(* Logix 5000 project; controller DC01 vendor 1 type 14 code 165 rev 32.12; software revision 32.04; part 9 of 13 *)
(* tags used below, declared in another part *)
   Always_Off : BOOL;
   Break_1stStation : BOOL;
   Break_LineWide : BOOL;
   Break_WorkCenter : BOOL;
   Break_Workstation : BOOL;
   FaultExists : CONTROL;
   LN03_MainLine_MSG : MESSAGE;   // Data Messages From Assembly Line 3 To Data Concentrator 1
   Local_Timer : TIMER[30];
   ONS_0 : DINT;
   Scheduled_Units_Buffer : DINT;
   Shift_Reset : BOOL;
   Shift_Reset_ONS : BOOL;
   LN02_Schedule : UDT_Current_Status;
   LN03_1st_Station_Break_Code : DINT;
   LN03_Additional_Break_Limit_Mins : DINT;
   LN03_Boxing_MNT : DINT;
   LN03_Console_MNT : DINT;
   LN03_Cooktop_MNT : DINT;
   LN03_Current_Shift_Duration_Mins : DINT;   // CURRENT SHIFT TOTAL MINUTES SCHEDULED
   LN03_Current_Shift_Duration_wBreaks_Mins : DINT;
   LN03_DC_Controlled_Theoretical_Units : BOOL;
   LN03_Door_MNT : DINT;
   LN03_FPY : REAL;
   LN03_FrontFrame_MNT : DINT;
   LN03_Ignition_NewSNModel : BOOL[32];
   LN03_Ignition_SNModelMSG : STRING[5];
   LN03_LeakTest_MNT : DINT;
   LN03_MachineOverAll_MNT : DINT;
   LN03_Main_Messages : DINT[250];
   LN03_MainBack_MNT : DINT;
   LN03_Messages_Barcode_SNModel : Barcode_SNModel;
   LN03_OT_Shift_Break_In_Minutes : DINT;
   LN03_OvenCavity_MNT : DINT;
   LN03_Schedule : UDT_Current_Status;
   LN03_Schedule_Cycle_Timer : TIMER;   // UNIT CYCLE ( TAKT TIME ) TIMER
   LN03_Schedule_Max_Break_Duration : DINT;
   LN03_Schedule_Max_Break_Timer : TIMER;
   LN03_Schedule_TAKT : REAL;
   LN03_SidePanels_MNT : DINT;
   LN03_Standard_Shift_Break_In_Minutes : DINT;
   LN03_StorageDrawer_MNT : DINT;
   LN03_Test_MNT : DINT;
   LN03_Theoretical_Units_Counter : COUNTER;   // CURRENT NUMBER OF UNITS THAT SHOULD BE BUILT
   LN03_Theoretical_Units_Counter_ONS : BOOL;
   LN03_Units_for_repair : DINT;
   LN03_Wiring_MNT : DINT;
   LN03ECM01 : DINT;
   LN03ECM02 : DINT;
   LN03ECM03 : DINT;
   LN03ECM04 : DINT;
   LN03ECM06 : DINT;
   LN03EDM04 : DINT;
   LN03EEM01 : DINT;
   LN03EES02 : DINT;
   LN03EES03 : DINT;
   LN03EES04 : DINT;
   LN03EGM01 : DINT;
   LN03EGM02 : DINT;
   LN03EHM01 : DINT;
   LN03NAS01 : DINT;
   LN03NAS02 : DINT;
   LN03NAS03 : DINT;
   LN03NAS04 : DINT;
   LN03NBS03 : DINT;
   LN03NCS01 : DINT;
   LN03NCS02 : DINT;
   LN03NCS03 : DINT;
   LN03NCS04 : DINT;
   LN03NCS05 : DINT;
   LN03NFS01 : DINT;
   LN03NFS03 : DINT;
   LN03SBS01 : DINT;
   LN03SBS02 : DINT;
   LN03SBS03 : DINT;
   LN03SCS03 : DINT;
   LN03SES01 : DINT;
   LN03SFS01 : DINT;
   LN03SFS02 : DINT;
   LN03SFS03 : DINT;
   LN03SFS04 : DINT;
   LN03WAM01 : DINT;
   LN03WBM01 : DINT;
   LN03WBM02 : DINT;
   LN03WCM02 : DINT;
   LN03WCM03 : DINT;
   LN03WCM04 : DINT;
   LN03WCM05 : DINT;
   LN03WDM01 : DINT;
   LN03WDM02 : DINT;
   LN03WDM03 : DINT;
   LN03WDM04 : DINT;
   LN03WDM05 : DINT;
   LN03WEM01 : DINT;
   LN03WEM02 : DINT;
   LN03WFM01 : DINT;
   LN03WFM02 : DINT;
   LN03WFM03 : DINT;
   LN03WFM04 : DINT;
   LN03WFM05 : DINT;
   LN03WFM06 : DINT;
   LN03WGM01 : DINT;
(* LN03, continued *)

ROUTINE R02_CurrentShift_Calcs   (* ladder *)
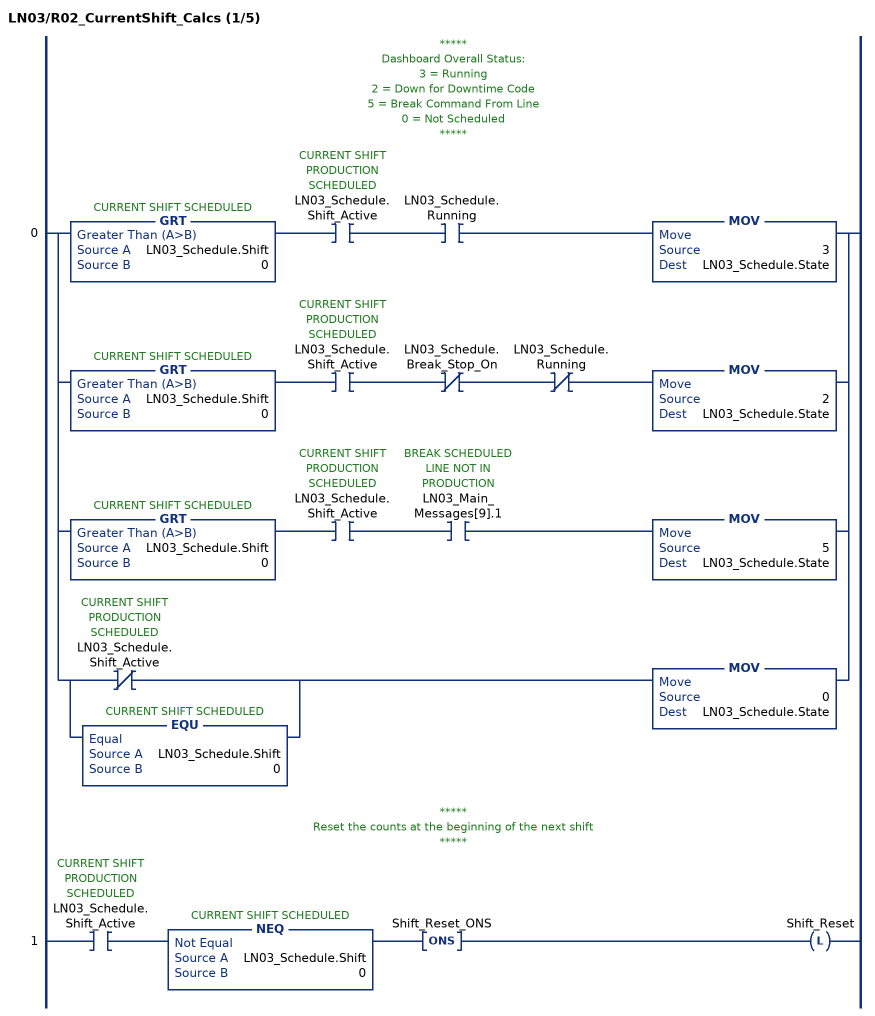
   // *****
   // Dashboard Overall Status:
   // 3 = Running
   // 2 = Down for Downtime Code
   // 5 = Break Command From Line
   // 0 = Not Scheduled
   // *****
   0: [GRT(LN03_Schedule.Shift,0) XIC(LN03_Schedule.Shift_Active) XIC(LN03_Schedule.Running) MOV(3,LN03_Schedule.State) ,GRT(LN03_Schedule.Shift,0) XIC(LN03_Schedule.Shift_Active) XIO(LN03_Schedule.Break_Stop_On) XIO(LN03_Schedule.Running) MOV(2,LN03_Schedule.State) ,GRT(LN03_Schedule.Shift,0) XIC(LN03_Schedule.Shift_Active) XIC(LN03_Main_Messages[9].1) MOV(5,LN03_Schedule.State) ,[XIO(LN03_Schedule.Shift_Active) ,EQU(LN03_Schedule.Shift,0) ] MOV(0,LN03_Schedule.State) ];
   // *****
   // Reset the counts at the beginning of the next shift
   // *****
   1: XIC(LN03_Schedule.Shift_Active)NEQ(LN03_Schedule.Shift,0)ONS(Shift_Reset_ONS)OTL(Shift_Reset);
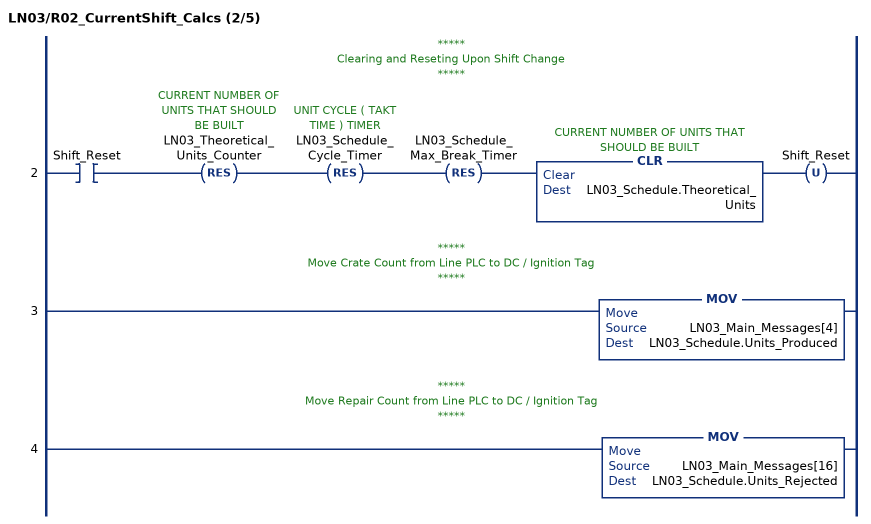
   // *****
   // Clearing and Reseting Upon Shift Change
   // *****
   2: XIC(Shift_Reset)RES(LN03_Theoretical_Units_Counter)RES(LN03_Schedule_Cycle_Timer)RES(LN03_Schedule_Max_Break_Timer)CLR(LN03_Schedule.Theoretical_Units)OTU(Shift_Reset);
   // *****
   // Move Crate Count from Line PLC to DC / Ignition Tag
   // *****
   3: MOV(LN03_Main_Messages[4],LN03_Schedule.Units_Produced);
   // *****
   // Move Repair Count from Line PLC to DC / Ignition Tag
   // *****
   4: MOV(LN03_Main_Messages[16],LN03_Schedule.Units_Rejected);
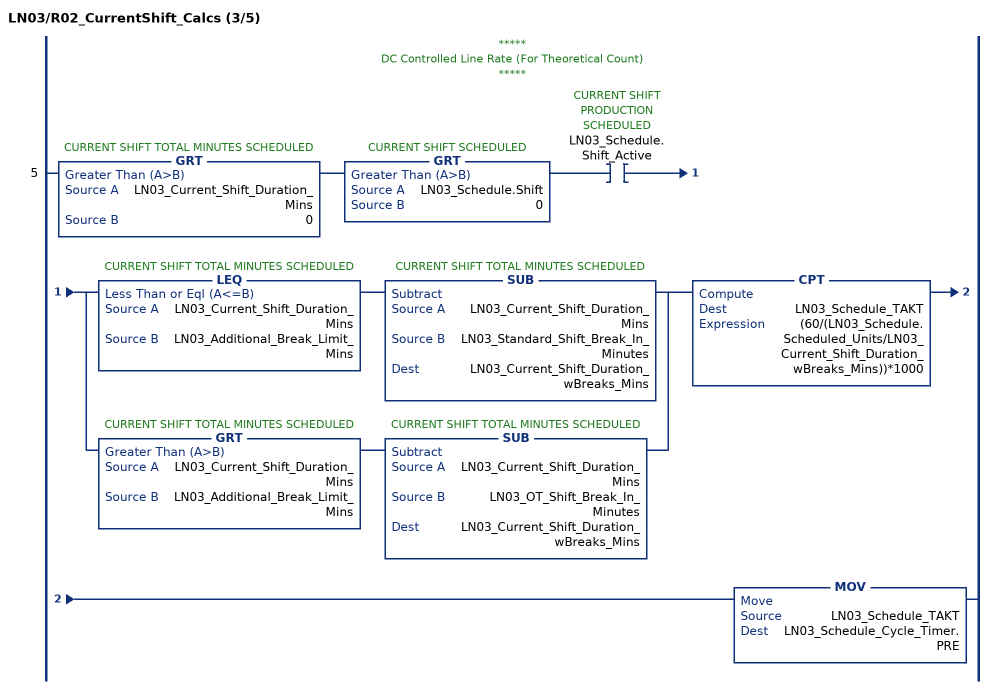
   // *****
   // DC Controlled Line Rate (For Theoretical Count)
   // *****
   5: GRT(LN03_Current_Shift_Duration_Mins,0)GRT(LN03_Schedule.Shift,0)XIC(LN03_Schedule.Shift_Active)[LEQ(LN03_Current_Shift_Duration_Mins,LN03_Additional_Break_Limit_Mins) SUB(LN03_Current_Shift_Duration_Mins,LN03_Standard_Shift_Break_In_Minutes,LN03_Current_Shift_Duration_wBreaks_Mins) ,GRT(LN03_Current_Shift_Duration_Mins,LN03_Additional_Break_Limit_Mins) SUB(LN03_Current_Shift_Duration_Mins,LN03_OT_Shift_Break_In_Minutes,LN03_Current_Shift_Duration_wBreaks_Mins) ]CPT(LN03_Schedule_TAKT,(60/(LN03_Schedule.Scheduled_Units/LN03_Current_Shift_Duration_wBreaks_Mins))*1000)MOV(LN03_Schedule_TAKT,LN03_Schedule_Cycle_Timer.PRE);
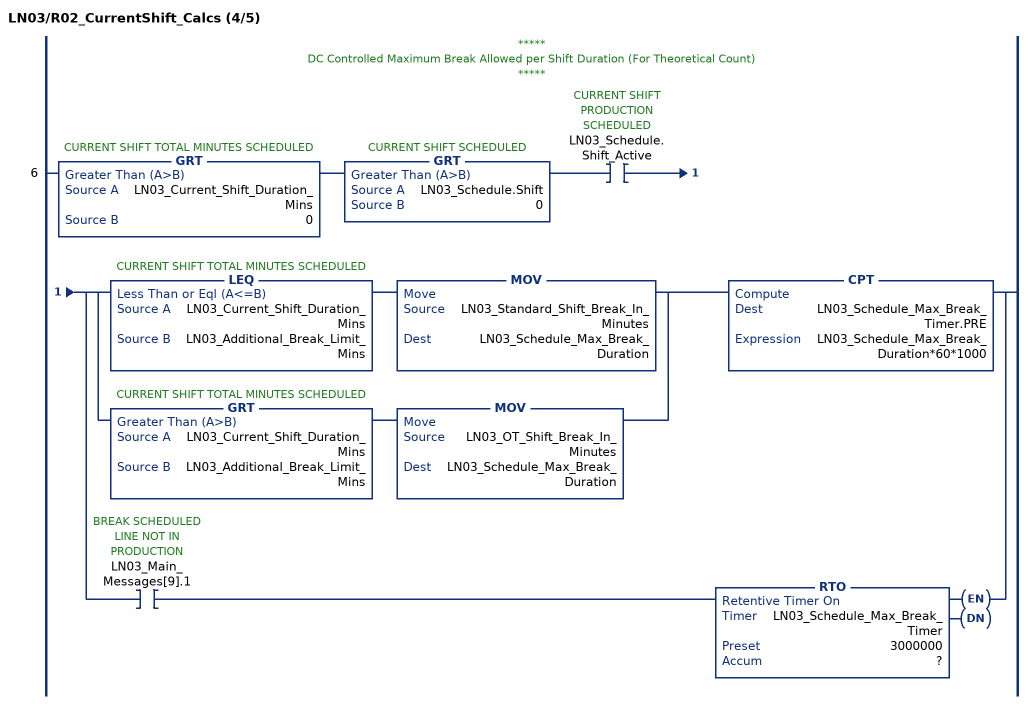
   // *****
   // DC Controlled Maximum Break Allowed per Shift Duration (For Theoretical Count)
   // *****
   6: GRT(LN03_Current_Shift_Duration_Mins,0)GRT(LN03_Schedule.Shift,0)XIC(LN03_Schedule.Shift_Active)[[LEQ(LN03_Current_Shift_Duration_Mins,LN03_Additional_Break_Limit_Mins) MOV(LN03_Standard_Shift_Break_In_Minutes,LN03_Schedule_Max_Break_Duration) ,GRT(LN03_Current_Shift_Duration_Mins,LN03_Additional_Break_Limit_Mins) MOV(LN03_OT_Shift_Break_In_Minutes,LN03_Schedule_Max_Break_Duration) ] CPT(LN03_Schedule_Max_Break_Timer.PRE,LN03_Schedule_Max_Break_Duration*60*1000) ,XIC(LN03_Main_Messages[9].1) RTO(LN03_Schedule_Max_Break_Timer,?,?) ];
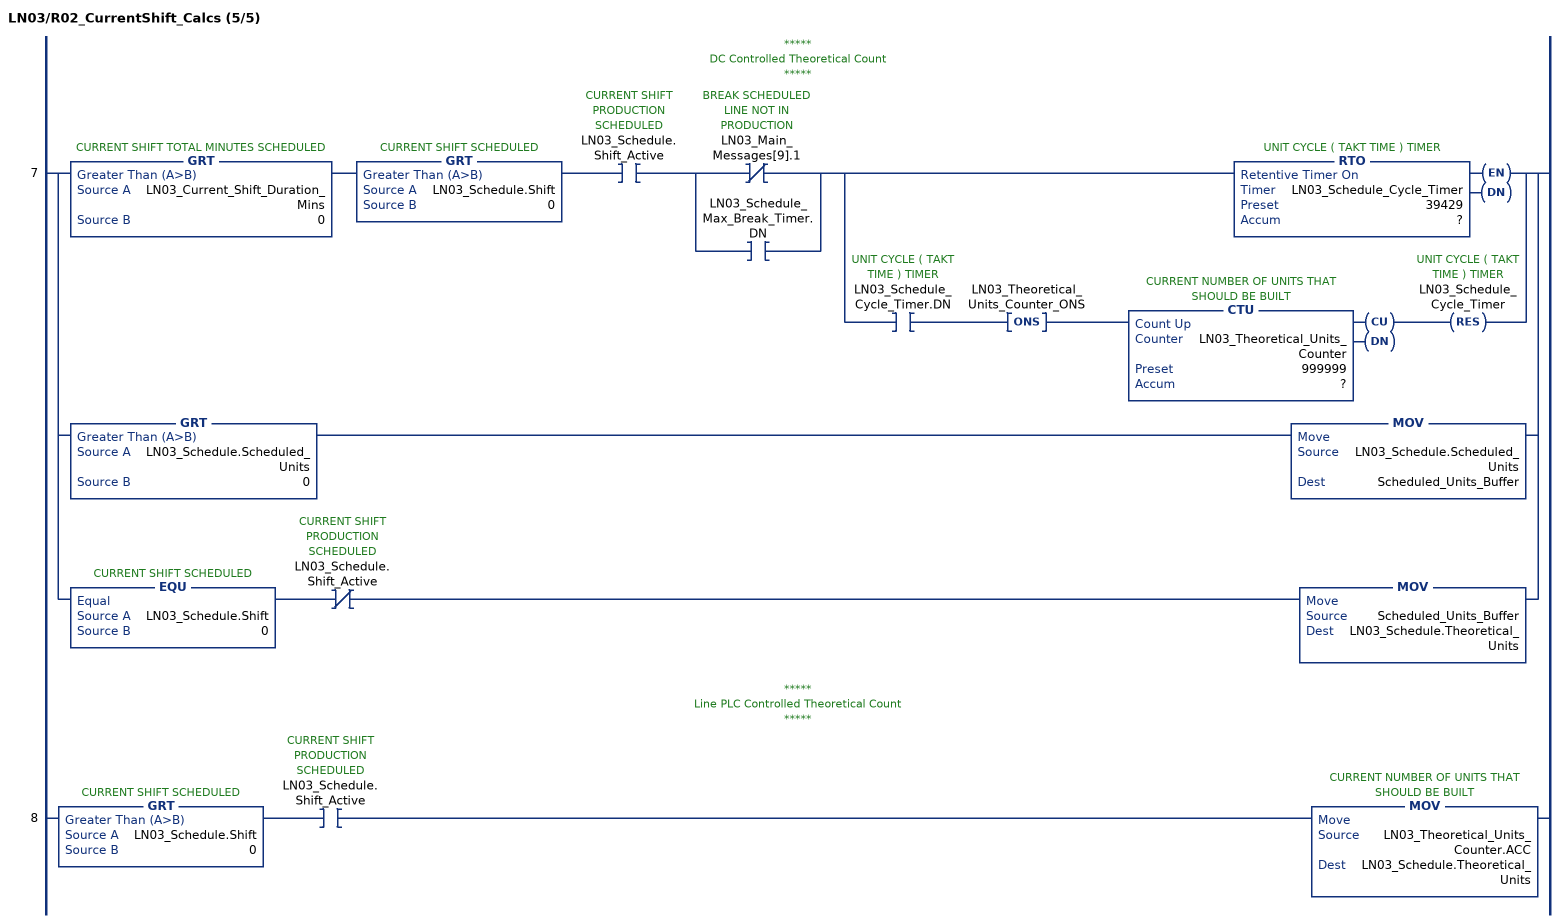
   // *****
   // DC Controlled Theoretical Count
   // *****
   7: [GRT(LN03_Current_Shift_Duration_Mins,0) GRT(LN03_Schedule.Shift,0) XIC(LN03_Schedule.Shift_Active) [XIO(LN03_Main_Messages[9].1) ,XIC(LN03_Schedule_Max_Break_Timer.DN) ] [RTO(LN03_Schedule_Cycle_Timer,?,?) ,XIC(LN03_Schedule_Cycle_Timer.DN) ONS(LN03_Theoretical_Units_Counter_ONS) CTU(LN03_Theoretical_Units_Counter,?,?) RES(LN03_Schedule_Cycle_Timer) ] ,GRT(LN03_Schedule.Scheduled_Units,0) MOV(LN03_Schedule.Scheduled_Units,Scheduled_Units_Buffer) ,EQU(LN03_Schedule.Shift,0) XIO(LN03_Schedule.Shift_Active) MOV(Scheduled_Units_Buffer,LN03_Schedule.Theoretical_Units) ];
   // *****
   // Line PLC Controlled Theoretical Count
   // *****
   8: GRT(LN03_Schedule.Shift,0)XIC(LN03_Schedule.Shift_Active)MOV(LN03_Theoretical_Units_Counter.ACC,LN03_Schedule.Theoretical_Units);
END_ROUTINE

ROUTINE R03_DataFromLines   (* ladder *)
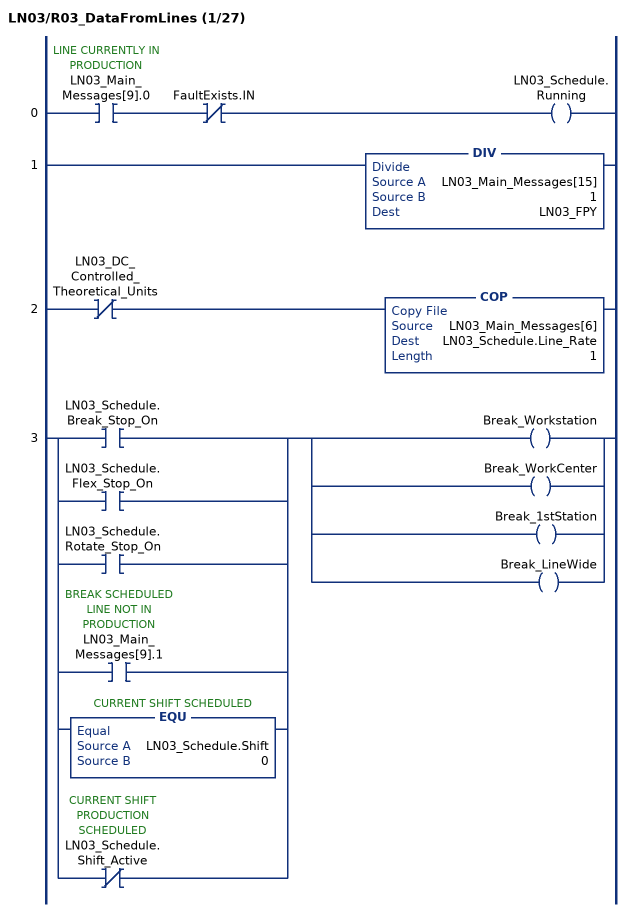
   0: XIC(LN03_Main_Messages[9].0)XIO(FaultExists.IN)OTE(LN03_Schedule.Running);
   1: DIV(LN03_Main_Messages[15],1,LN03_FPY);
   2: XIO(LN03_DC_Controlled_Theoretical_Units)COP(LN03_Main_Messages[6],LN03_Schedule.Line_Rate,1);
   3: [XIC(LN03_Schedule.Break_Stop_On) ,XIC(LN03_Schedule.Flex_Stop_On) ,XIC(LN03_Schedule.Rotate_Stop_On) ,XIC(LN03_Main_Messages[9].1) ,EQU(LN03_Schedule.Shift,0) ,XIO(LN03_Schedule.Shift_Active) ][OTE(Break_Workstation) ,OTE(Break_WorkCenter) ,OTE(Break_1stStation) ,OTE(Break_LineWide) ];
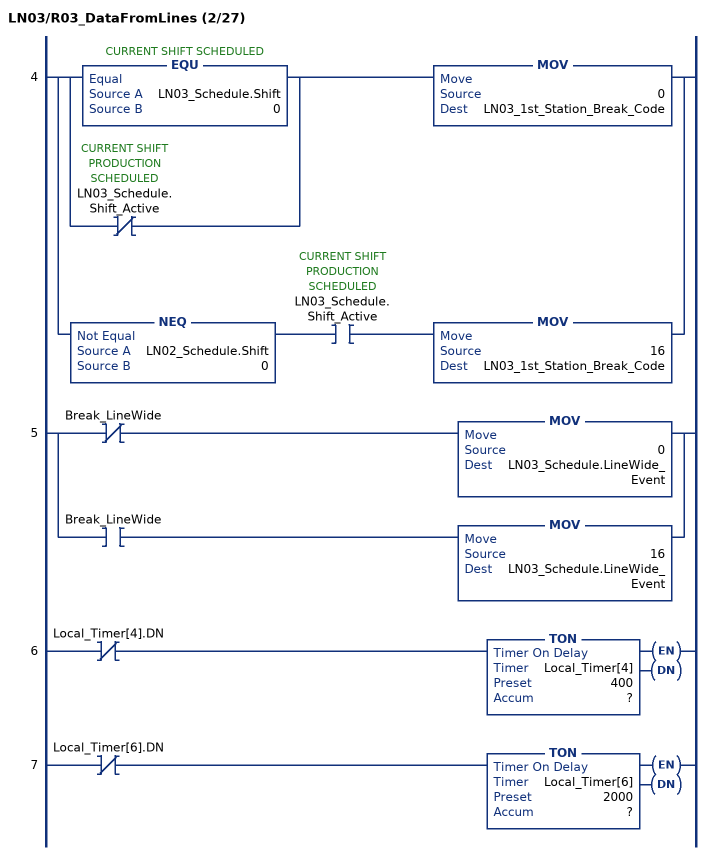
   4: [[EQU(LN03_Schedule.Shift,0) ,XIO(LN03_Schedule.Shift_Active) ] MOV(0,LN03_1st_Station_Break_Code) ,NEQ(LN02_Schedule.Shift,0) XIC(LN03_Schedule.Shift_Active) MOV(16,LN03_1st_Station_Break_Code) ];
   5: [XIO(Break_LineWide) MOV(0,LN03_Schedule.LineWide_Event) ,XIC(Break_LineWide) MOV(16,LN03_Schedule.LineWide_Event) ];
   6: XIO(Local_Timer[4].DN)TON(Local_Timer[4],?,?);
   7: XIO(Local_Timer[6].DN)TON(Local_Timer[6],?,?);
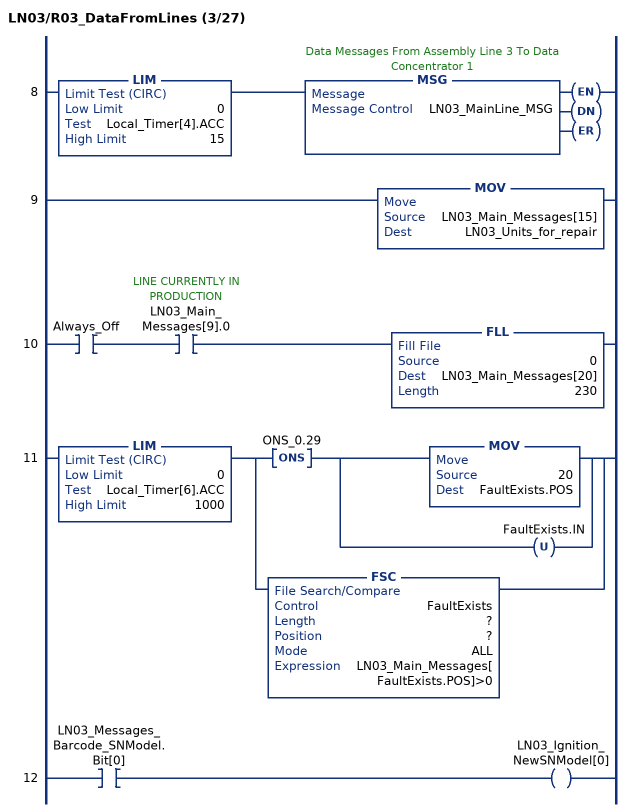
   8: LIM(0,Local_Timer[4].ACC,15)MSG(LN03_MainLine_MSG);
   9: MOV(LN03_Main_Messages[15],LN03_Units_for_repair);
   10: XIC(Always_Off)XIC(LN03_Main_Messages[9].0)FLL(0,LN03_Main_Messages[20],230);
   11: LIM(0,Local_Timer[6].ACC,1000)[ONS(ONS_0.29) [MOV(20,FaultExists.POS) ,OTU(FaultExists.IN) ] ,FSC(FaultExists,?,?,ALL,LN03_Main_Messages[FaultExists.POS]>0) ];
   12: XIC(LN03_Messages_Barcode_SNModel.Bit[0])OTE(LN03_Ignition_NewSNModel[0]);
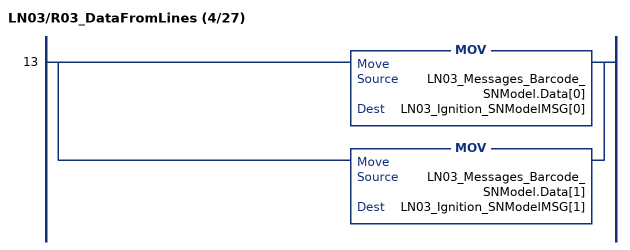
   13: [MOV(LN03_Messages_Barcode_SNModel.Data[0],LN03_Ignition_SNModelMSG[0]) ,MOV(LN03_Messages_Barcode_SNModel.Data[1],LN03_Ignition_SNModelMSG[1]) ];
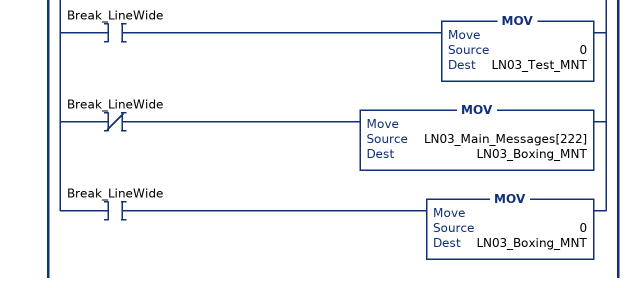
   14: [XIO(Break_LineWide) MOV(LN03_Main_Messages[20],LN03_MachineOverAll_MNT) ,XIC(Break_LineWide) MOV(0,LN03_MachineOverAll_MNT) ,XIO(Break_LineWide) MOV(LN03_Main_Messages[21],LN03_FrontFrame_MNT) ,XIC(Break_LineWide) MOV(0,LN03_FrontFrame_MNT) ,XIO(Break_LineWide) MOV(LN03_Main_Messages[22],LN03_OvenCavity_MNT) ,XIC(Break_LineWide) MOV(0,LN03_OvenCavity_MNT) ,XIO(Break_LineWide) MOV(LN03_Main_Messages[23],LN03_MainBack_MNT) ,XIC(Break_LineWide) MOV(0,LN03_MainBack_MNT) ,XIO(Break_LineWide) MOV(LN03_Main_Messages[24],LN03_SidePanels_MNT) ,XIC(Break_LineWide) MOV(0,LN03_SidePanels_MNT) ,XIO(Break_LineWide) MOV(LN03_Main_Messages[25],LN03_Console_MNT) ,XIC(Break_LineWide) MOV(0,LN03_Console_MNT) ,XIO(Break_LineWide) MOV(LN03_Main_Messages[26],LN03_Cooktop_MNT) ,XIC(Break_LineWide) MOV(0,LN03_Cooktop_MNT) ,XIO(Break_LineWide) MOV(LN03_Main_Messages[27],LN03_LeakTest_MNT) ,XIC(Break_LineWide) MOV(0,LN03_LeakTest_MNT) ,XIO(Break_LineWide) MOV(LN03_Main_Messages[28],LN03_Wiring_MNT) ,XIC(Break_LineWide) MOV(0,LN03_Wiring_MNT) ,XIO(Break_LineWide) MOV(LN03_Main_Messages[29],LN03_StorageDrawer_MNT) ,XIC(Break_LineWide) MOV(0,LN03_StorageDrawer_MNT) ,XIO(Break_LineWide) MOV(LN03_Main_Messages[220],LN03_Door_MNT) ,XIC(Break_LineWide) MOV(0,LN03_Door_MNT) ,XIO(Break_LineWide) MOV(LN03_Main_Messages[221],LN03_Test_MNT) ,XIC(Break_LineWide) MOV(0,LN03_Test_MNT) ,XIO(Break_LineWide) MOV(LN03_Main_Messages[222],LN03_Boxing_MNT) ,XIC(Break_LineWide) MOV(0,LN03_Boxing_MNT) ];
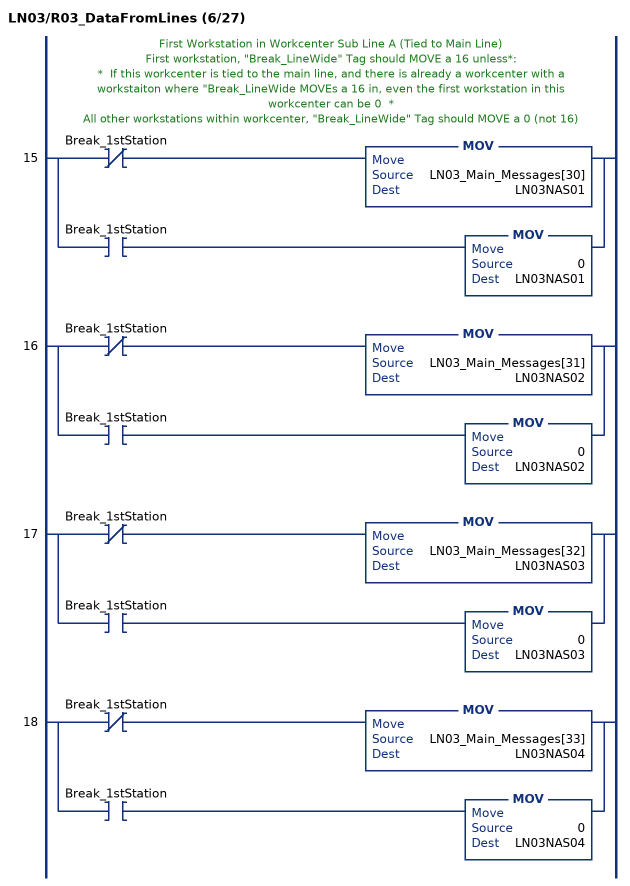
   // First Workstation in Workcenter Sub Line A (Tied to Main Line)
   // First workstation, "Break_LineWide" Tag should MOVE a 16 unless*:
   // *  If this workcenter is tied to the main line, and there is already a workcenter with a workstaiton where "Break_LineWide MOVEs a 16 in, even the first workstation in this workcenter can be 0  *
   // All other workstations within workcenter, "Break_LineWide" Tag should MOVE a 0 (not 16)
   15: [XIO(Break_1stStation) MOV(LN03_Main_Messages[30],LN03NAS01) ,XIC(Break_1stStation) MOV(0,LN03NAS01) ];
   16: [XIO(Break_1stStation) MOV(LN03_Main_Messages[31],LN03NAS02) ,XIC(Break_1stStation) MOV(0,LN03NAS02) ];
   17: [XIO(Break_1stStation) MOV(LN03_Main_Messages[32],LN03NAS03) ,XIC(Break_1stStation) MOV(0,LN03NAS03) ];
   18: [XIO(Break_1stStation) MOV(LN03_Main_Messages[33],LN03NAS04) ,XIC(Break_1stStation) MOV(0,LN03NAS04) ];
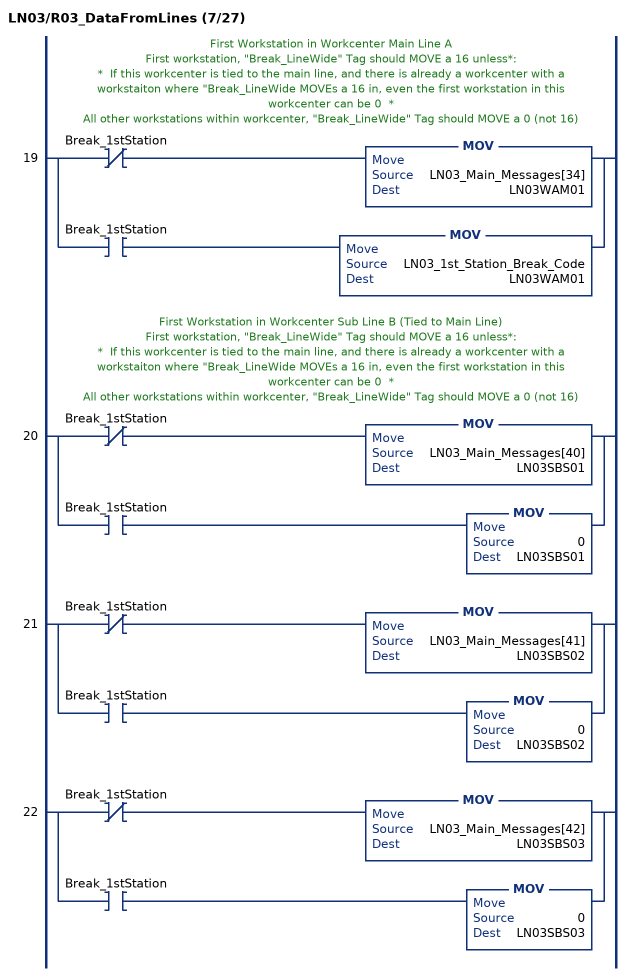
   // First Workstation in Workcenter Main Line A
   // First workstation, "Break_LineWide" Tag should MOVE a 16 unless*:
   // *  If this workcenter is tied to the main line, and there is already a workcenter with a workstaiton where "Break_LineWide MOVEs a 16 in, even the first workstation in this workcenter can be 0  *
   // All other workstations within workcenter, "Break_LineWide" Tag should MOVE a 0 (not 16)
   19: [XIO(Break_1stStation) MOV(LN03_Main_Messages[34],LN03WAM01) ,XIC(Break_1stStation) MOV(LN03_1st_Station_Break_Code,LN03WAM01) ];
   // First Workstation in Workcenter Sub Line B (Tied to Main Line)
   // First workstation, "Break_LineWide" Tag should MOVE a 16 unless*:
   // *  If this workcenter is tied to the main line, and there is already a workcenter with a workstaiton where "Break_LineWide MOVEs a 16 in, even the first workstation in this workcenter can be 0  *
   // All other workstations within workcenter, "Break_LineWide" Tag should MOVE a 0 (not 16)
   20: [XIO(Break_1stStation) MOV(LN03_Main_Messages[40],LN03SBS01) ,XIC(Break_1stStation) MOV(0,LN03SBS01) ];
   21: [XIO(Break_1stStation) MOV(LN03_Main_Messages[41],LN03SBS02) ,XIC(Break_1stStation) MOV(0,LN03SBS02) ];
   22: [XIO(Break_1stStation) MOV(LN03_Main_Messages[42],LN03SBS03) ,XIC(Break_1stStation) MOV(0,LN03SBS03) ];
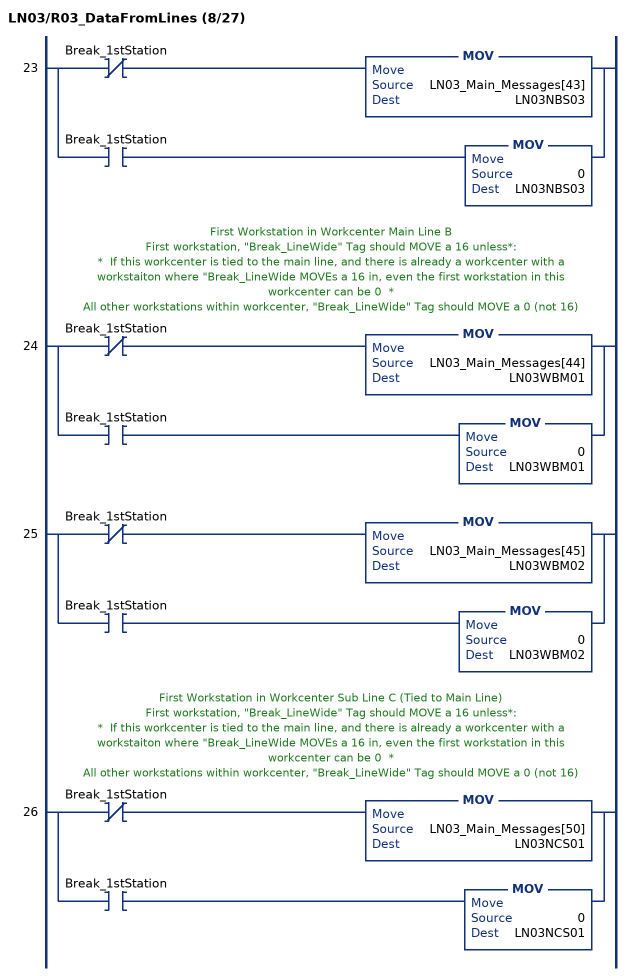
   23: [XIO(Break_1stStation) MOV(LN03_Main_Messages[43],LN03NBS03) ,XIC(Break_1stStation) MOV(0,LN03NBS03) ];
   // First Workstation in Workcenter Main Line B
   // First workstation, "Break_LineWide" Tag should MOVE a 16 unless*:
   // *  If this workcenter is tied to the main line, and there is already a workcenter with a workstaiton where "Break_LineWide MOVEs a 16 in, even the first workstation in this workcenter can be 0  *
   // All other workstations within workcenter, "Break_LineWide" Tag should MOVE a 0 (not 16)
   24: [XIO(Break_1stStation) MOV(LN03_Main_Messages[44],LN03WBM01) ,XIC(Break_1stStation) MOV(0,LN03WBM01) ];
   25: [XIO(Break_1stStation) MOV(LN03_Main_Messages[45],LN03WBM02) ,XIC(Break_1stStation) MOV(0,LN03WBM02) ];
   // First Workstation in Workcenter Sub Line C (Tied to Main Line)
   // First workstation, "Break_LineWide" Tag should MOVE a 16 unless*:
   // *  If this workcenter is tied to the main line, and there is already a workcenter with a workstaiton where "Break_LineWide MOVEs a 16 in, even the first workstation in this workcenter can be 0  *
   // All other workstations within workcenter, "Break_LineWide" Tag should MOVE a 0 (not 16)
   26: [XIO(Break_1stStation) MOV(LN03_Main_Messages[50],LN03NCS01) ,XIC(Break_1stStation) MOV(0,LN03NCS01) ];
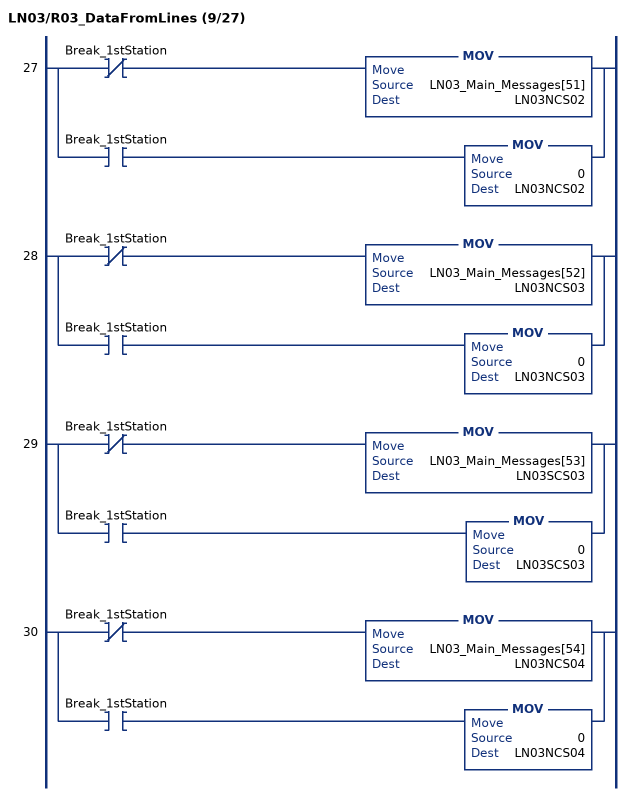
   27: [XIO(Break_1stStation) MOV(LN03_Main_Messages[51],LN03NCS02) ,XIC(Break_1stStation) MOV(0,LN03NCS02) ];
   28: [XIO(Break_1stStation) MOV(LN03_Main_Messages[52],LN03NCS03) ,XIC(Break_1stStation) MOV(0,LN03NCS03) ];
   29: [XIO(Break_1stStation) MOV(LN03_Main_Messages[53],LN03SCS03) ,XIC(Break_1stStation) MOV(0,LN03SCS03) ];
   30: [XIO(Break_1stStation) MOV(LN03_Main_Messages[54],LN03NCS04) ,XIC(Break_1stStation) MOV(0,LN03NCS04) ];
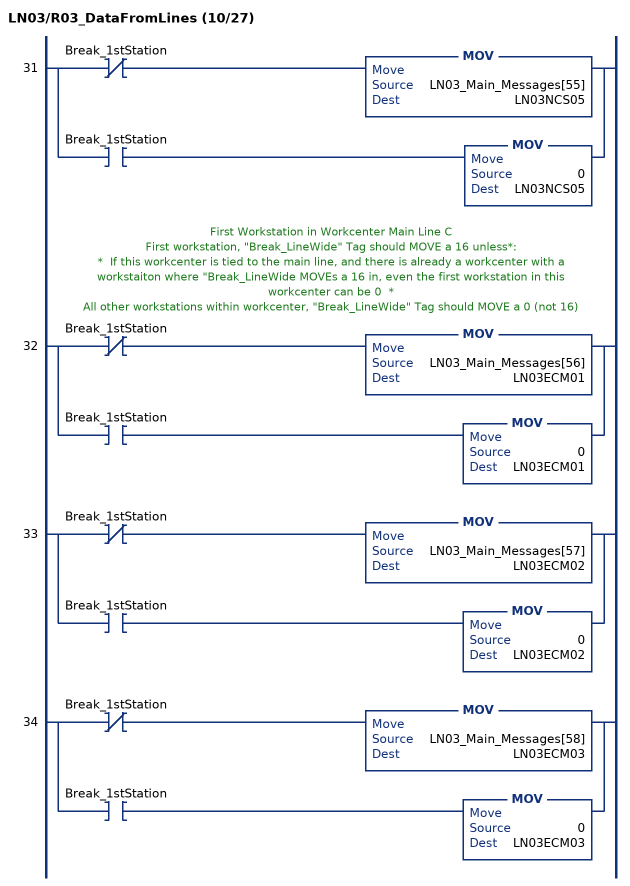
   31: [XIO(Break_1stStation) MOV(LN03_Main_Messages[55],LN03NCS05) ,XIC(Break_1stStation) MOV(0,LN03NCS05) ];
   // First Workstation in Workcenter Main Line C
   // First workstation, "Break_LineWide" Tag should MOVE a 16 unless*:
   // *  If this workcenter is tied to the main line, and there is already a workcenter with a workstaiton where "Break_LineWide MOVEs a 16 in, even the first workstation in this workcenter can be 0  *
   // All other workstations within workcenter, "Break_LineWide" Tag should MOVE a 0 (not 16)
   32: [XIO(Break_1stStation) MOV(LN03_Main_Messages[56],LN03ECM01) ,XIC(Break_1stStation) MOV(0,LN03ECM01) ];
   33: [XIO(Break_1stStation) MOV(LN03_Main_Messages[57],LN03ECM02) ,XIC(Break_1stStation) MOV(0,LN03ECM02) ];
   34: [XIO(Break_1stStation) MOV(LN03_Main_Messages[58],LN03ECM03) ,XIC(Break_1stStation) MOV(0,LN03ECM03) ];
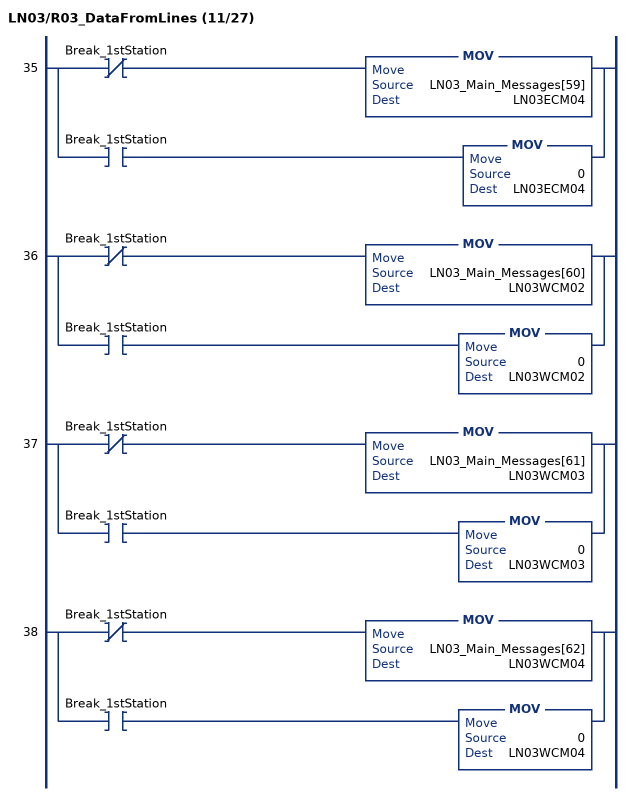
   35: [XIO(Break_1stStation) MOV(LN03_Main_Messages[59],LN03ECM04) ,XIC(Break_1stStation) MOV(0,LN03ECM04) ];
   36: [XIO(Break_1stStation) MOV(LN03_Main_Messages[60],LN03WCM02) ,XIC(Break_1stStation) MOV(0,LN03WCM02) ];
   37: [XIO(Break_1stStation) MOV(LN03_Main_Messages[61],LN03WCM03) ,XIC(Break_1stStation) MOV(0,LN03WCM03) ];
   38: [XIO(Break_1stStation) MOV(LN03_Main_Messages[62],LN03WCM04) ,XIC(Break_1stStation) MOV(0,LN03WCM04) ];
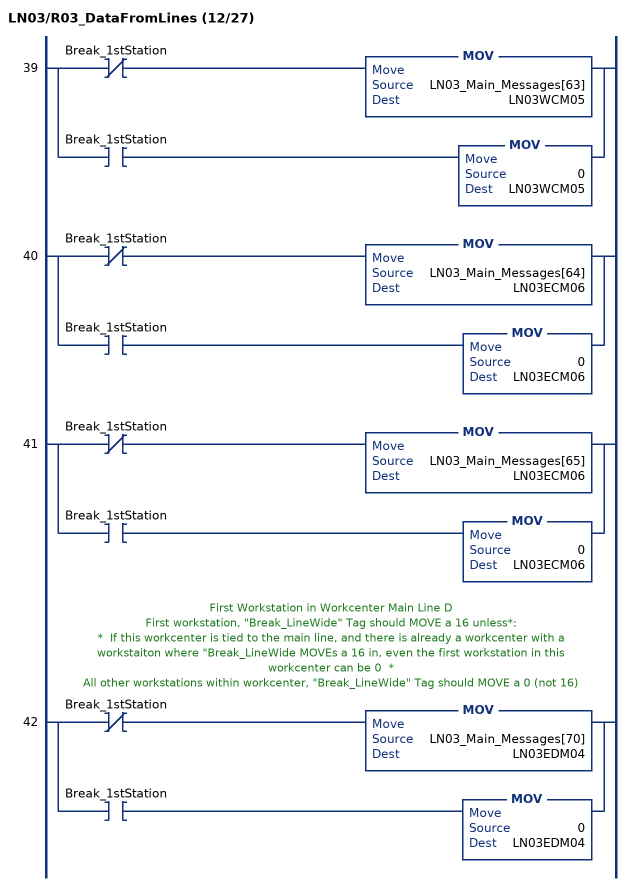
   39: [XIO(Break_1stStation) MOV(LN03_Main_Messages[63],LN03WCM05) ,XIC(Break_1stStation) MOV(0,LN03WCM05) ];
   40: [XIO(Break_1stStation) MOV(LN03_Main_Messages[64],LN03ECM06) ,XIC(Break_1stStation) MOV(0,LN03ECM06) ];
   41: [XIO(Break_1stStation) MOV(LN03_Main_Messages[65],LN03ECM06) ,XIC(Break_1stStation) MOV(0,LN03ECM06) ];
   // First Workstation in Workcenter Main Line D
   // First workstation, "Break_LineWide" Tag should MOVE a 16 unless*:
   // *  If this workcenter is tied to the main line, and there is already a workcenter with a workstaiton where "Break_LineWide MOVEs a 16 in, even the first workstation in this workcenter can be 0  *
   // All other workstations within workcenter, "Break_LineWide" Tag should MOVE a 0 (not 16)
   42: [XIO(Break_1stStation) MOV(LN03_Main_Messages[70],LN03EDM04) ,XIC(Break_1stStation) MOV(0,LN03EDM04) ];
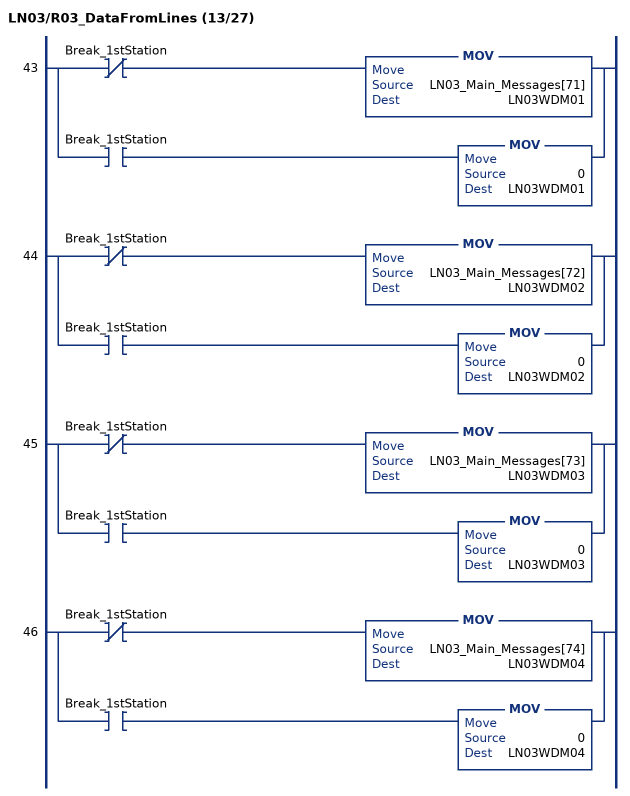
   43: [XIO(Break_1stStation) MOV(LN03_Main_Messages[71],LN03WDM01) ,XIC(Break_1stStation) MOV(0,LN03WDM01) ];
   44: [XIO(Break_1stStation) MOV(LN03_Main_Messages[72],LN03WDM02) ,XIC(Break_1stStation) MOV(0,LN03WDM02) ];
   45: [XIO(Break_1stStation) MOV(LN03_Main_Messages[73],LN03WDM03) ,XIC(Break_1stStation) MOV(0,LN03WDM03) ];
   46: [XIO(Break_1stStation) MOV(LN03_Main_Messages[74],LN03WDM04) ,XIC(Break_1stStation) MOV(0,LN03WDM04) ];
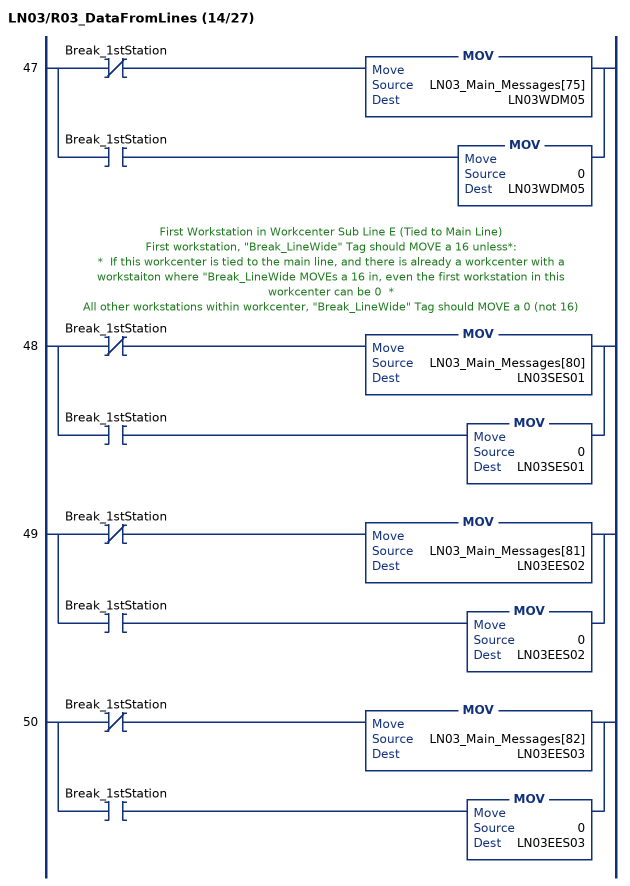
   47: [XIO(Break_1stStation) MOV(LN03_Main_Messages[75],LN03WDM05) ,XIC(Break_1stStation) MOV(0,LN03WDM05) ];
   // First Workstation in Workcenter Sub Line E (Tied to Main Line)
   // First workstation, "Break_LineWide" Tag should MOVE a 16 unless*:
   // *  If this workcenter is tied to the main line, and there is already a workcenter with a workstaiton where "Break_LineWide MOVEs a 16 in, even the first workstation in this workcenter can be 0  *
   // All other workstations within workcenter, "Break_LineWide" Tag should MOVE a 0 (not 16)
   48: [XIO(Break_1stStation) MOV(LN03_Main_Messages[80],LN03SES01) ,XIC(Break_1stStation) MOV(0,LN03SES01) ];
   49: [XIO(Break_1stStation) MOV(LN03_Main_Messages[81],LN03EES02) ,XIC(Break_1stStation) MOV(0,LN03EES02) ];
   50: [XIO(Break_1stStation) MOV(LN03_Main_Messages[82],LN03EES03) ,XIC(Break_1stStation) MOV(0,LN03EES03) ];
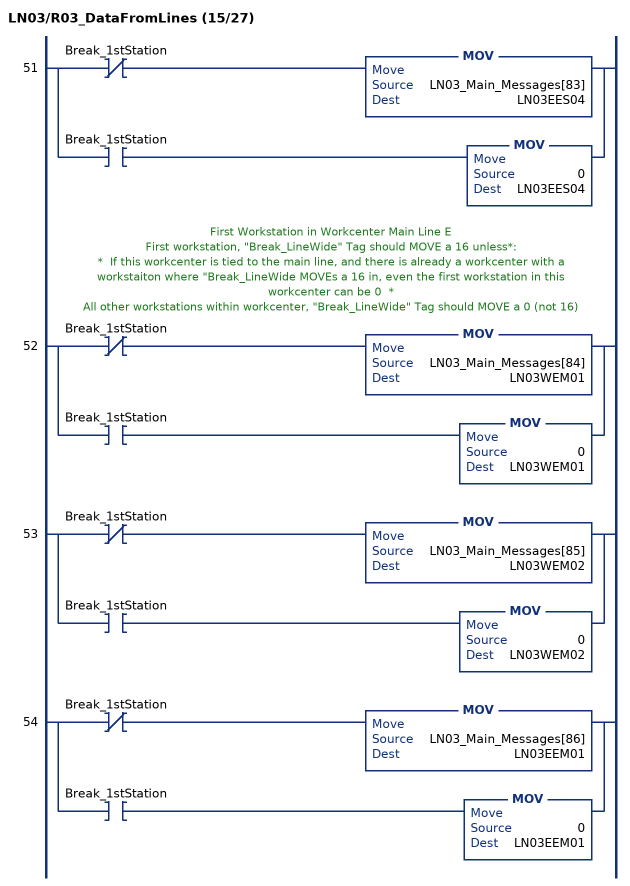
   51: [XIO(Break_1stStation) MOV(LN03_Main_Messages[83],LN03EES04) ,XIC(Break_1stStation) MOV(0,LN03EES04) ];
   // First Workstation in Workcenter Main Line E
   // First workstation, "Break_LineWide" Tag should MOVE a 16 unless*:
   // *  If this workcenter is tied to the main line, and there is already a workcenter with a workstaiton where "Break_LineWide MOVEs a 16 in, even the first workstation in this workcenter can be 0  *
   // All other workstations within workcenter, "Break_LineWide" Tag should MOVE a 0 (not 16)
   52: [XIO(Break_1stStation) MOV(LN03_Main_Messages[84],LN03WEM01) ,XIC(Break_1stStation) MOV(0,LN03WEM01) ];
   53: [XIO(Break_1stStation) MOV(LN03_Main_Messages[85],LN03WEM02) ,XIC(Break_1stStation) MOV(0,LN03WEM02) ];
   54: [XIO(Break_1stStation) MOV(LN03_Main_Messages[86],LN03EEM01) ,XIC(Break_1stStation) MOV(0,LN03EEM01) ];
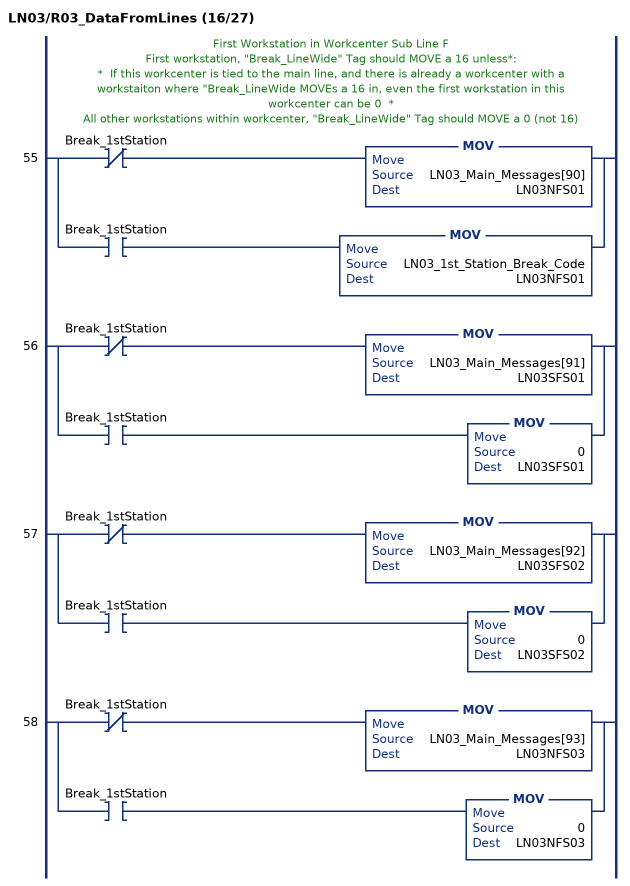
   // First Workstation in Workcenter Sub Line F
   // First workstation, "Break_LineWide" Tag should MOVE a 16 unless*:
   // *  If this workcenter is tied to the main line, and there is already a workcenter with a workstaiton where "Break_LineWide MOVEs a 16 in, even the first workstation in this workcenter can be 0  *
   // All other workstations within workcenter, "Break_LineWide" Tag should MOVE a 0 (not 16)
   55: [XIO(Break_1stStation) MOV(LN03_Main_Messages[90],LN03NFS01) ,XIC(Break_1stStation) MOV(LN03_1st_Station_Break_Code,LN03NFS01) ];
   56: [XIO(Break_1stStation) MOV(LN03_Main_Messages[91],LN03SFS01) ,XIC(Break_1stStation) MOV(0,LN03SFS01) ];
   57: [XIO(Break_1stStation) MOV(LN03_Main_Messages[92],LN03SFS02) ,XIC(Break_1stStation) MOV(0,LN03SFS02) ];
   58: [XIO(Break_1stStation) MOV(LN03_Main_Messages[93],LN03NFS03) ,XIC(Break_1stStation) MOV(0,LN03NFS03) ];
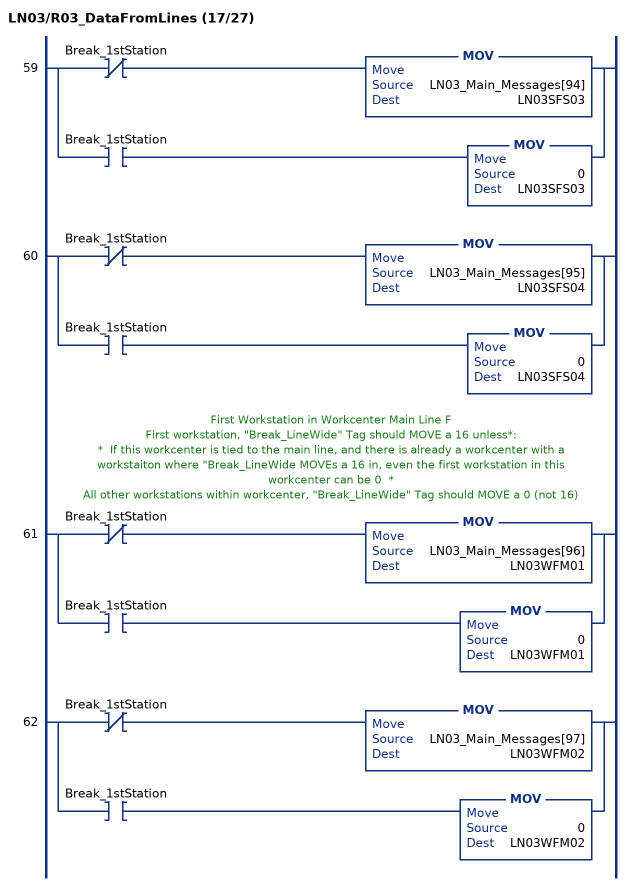
   59: [XIO(Break_1stStation) MOV(LN03_Main_Messages[94],LN03SFS03) ,XIC(Break_1stStation) MOV(0,LN03SFS03) ];
   60: [XIO(Break_1stStation) MOV(LN03_Main_Messages[95],LN03SFS04) ,XIC(Break_1stStation) MOV(0,LN03SFS04) ];
   // First Workstation in Workcenter Main Line F
   // First workstation, "Break_LineWide" Tag should MOVE a 16 unless*:
   // *  If this workcenter is tied to the main line, and there is already a workcenter with a workstaiton where "Break_LineWide MOVEs a 16 in, even the first workstation in this workcenter can be 0  *
   // All other workstations within workcenter, "Break_LineWide" Tag should MOVE a 0 (not 16)
   61: [XIO(Break_1stStation) MOV(LN03_Main_Messages[96],LN03WFM01) ,XIC(Break_1stStation) MOV(0,LN03WFM01) ];
   62: [XIO(Break_1stStation) MOV(LN03_Main_Messages[97],LN03WFM02) ,XIC(Break_1stStation) MOV(0,LN03WFM02) ];
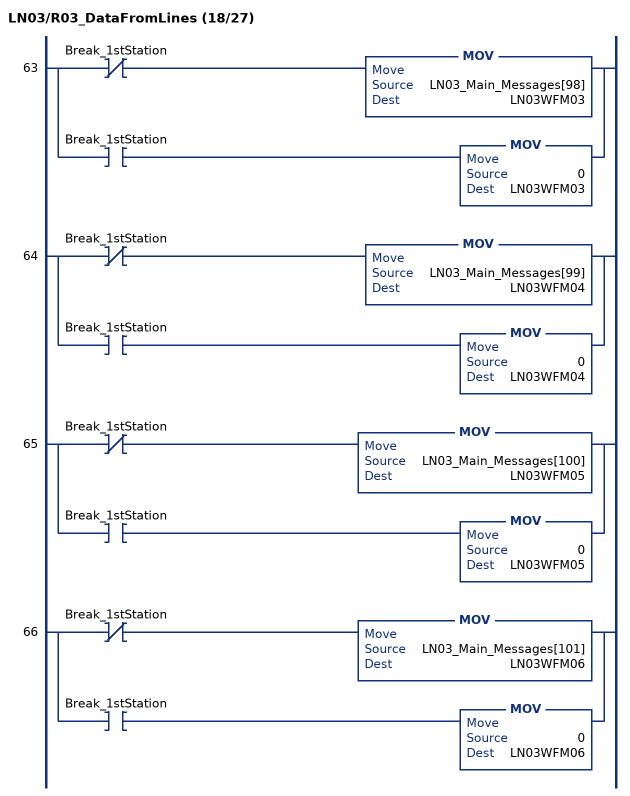
   63: [XIO(Break_1stStation) MOV(LN03_Main_Messages[98],LN03WFM03) ,XIC(Break_1stStation) MOV(0,LN03WFM03) ];
   64: [XIO(Break_1stStation) MOV(LN03_Main_Messages[99],LN03WFM04) ,XIC(Break_1stStation) MOV(0,LN03WFM04) ];
   65: [XIO(Break_1stStation) MOV(LN03_Main_Messages[100],LN03WFM05) ,XIC(Break_1stStation) MOV(0,LN03WFM05) ];
   66: [XIO(Break_1stStation) MOV(LN03_Main_Messages[101],LN03WFM06) ,XIC(Break_1stStation) MOV(0,LN03WFM06) ];
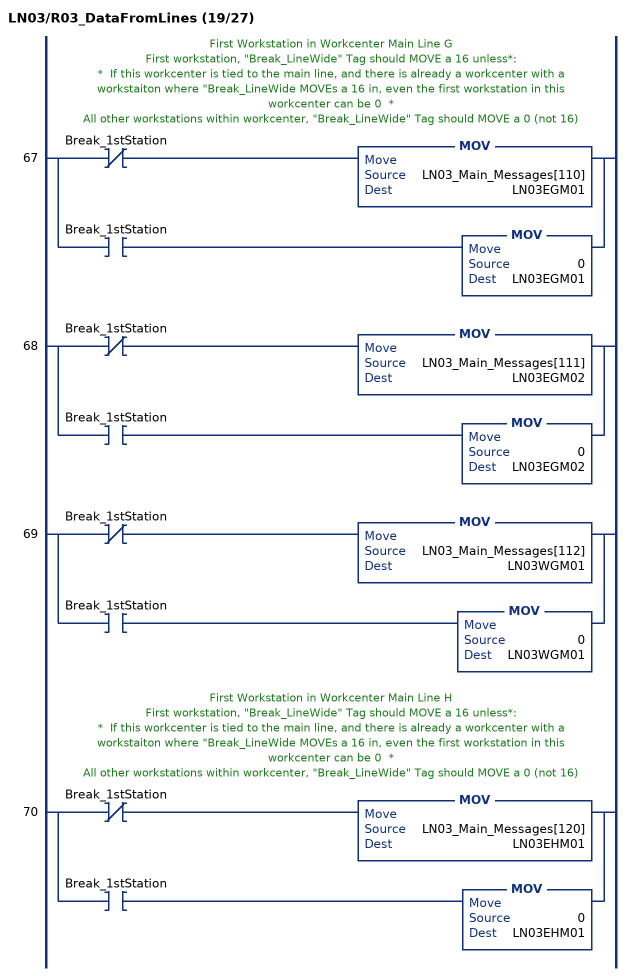
   // First Workstation in Workcenter Main Line G
   // First workstation, "Break_LineWide" Tag should MOVE a 16 unless*:
   // *  If this workcenter is tied to the main line, and there is already a workcenter with a workstaiton where "Break_LineWide MOVEs a 16 in, even the first workstation in this workcenter can be 0  *
   // All other workstations within workcenter, "Break_LineWide" Tag should MOVE a 0 (not 16)
   67: [XIO(Break_1stStation) MOV(LN03_Main_Messages[110],LN03EGM01) ,XIC(Break_1stStation) MOV(0,LN03EGM01) ];
   68: [XIO(Break_1stStation) MOV(LN03_Main_Messages[111],LN03EGM02) ,XIC(Break_1stStation) MOV(0,LN03EGM02) ];
   69: [XIO(Break_1stStation) MOV(LN03_Main_Messages[112],LN03WGM01) ,XIC(Break_1stStation) MOV(0,LN03WGM01) ];
   // First Workstation in Workcenter Main Line H
   // First workstation, "Break_LineWide" Tag should MOVE a 16 unless*:
   // *  If this workcenter is tied to the main line, and there is already a workcenter with a workstaiton where "Break_LineWide MOVEs a 16 in, even the first workstation in this workcenter can be 0  *
   // All other workstations within workcenter, "Break_LineWide" Tag should MOVE a 0 (not 16)
   70: [XIO(Break_1stStation) MOV(LN03_Main_Messages[120],LN03EHM01) ,XIC(Break_1stStation) MOV(0,LN03EHM01) ];
